FUNCTION_BLOCK pulse_
VAR_INPUT
END_VAR
VAR_OUTPUT
	out: BOOL;
END_VAR
VAR
END_VAR

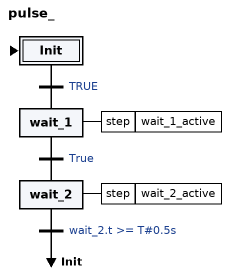
INITIAL_STEP Init:
END_STEP
TRANSITION FROM Init TO wait_1
    := TRUE;
END_TRANSITION
STEP wait_1:
    wait_1_active(N);  // step action
END_STEP
TRANSITION FROM wait_1 TO wait_2
    := True;
END_TRANSITION
STEP wait_2:
    wait_2_active(N);  // step action
END_STEP
TRANSITION FROM wait_2 TO Init
    := wait_2.t >= T#0.5s;
END_TRANSITION

ACTION wait_1_active:
out := True;
END_ACTION

ACTION wait_2_active:
out := False;
END_ACTION

END_FUNCTION_BLOCK

(* stored: Version 1.1.0.1, ProductVersion 3.1.4024.4
   POU pulse_: Id {79f948f9-33b9-4186-b2f6-cf9fc06ace38}, SpecialFunc None
   Action wait_1_active: Id {3c902b6f-af16-44aa-b1f8-c43933e60533}
   Action wait_2_active: Id {9c43a5df-47ba-4143-8393-150ef5ee3c8d} *)
